Universal Robots PolyScope program: Main3.urp

Program Main3 (installation=main2 directory=/programs createdIn=5.11.5.1010327 lastSavedIn=5.11.5.1010327 robotSerialNumber=20215500677)
Calibrated DH parameters: a=[0.000204, -0.239222, -0.391845, -0.000001, 0.000022, 0]; d=[0.162722, -355.808559, 353.37206, 2.570385, 0.099741, 0.099629]; alpha=[1.571124, 0.000988, 0.008295, 1.568963, -1.570303, 0]; deltaTheta=[0, -0.973091, 7.204745, 0.05153, 0, 0]
Robot Program (runOnlyOnce=true)
  MoveJ speed 60 deg/s, acceleration 80 deg/s^2 (useActiveTCP=true) feature=CubeFront
    Waypoint Clear: TCP in base x=-162.331 y=-451.249 z=327.15 mm, rx=0.0678 ry=2.1899 rz=-2.19 rad; joints [27.656, -90.853, 115.036, 43.322, 49.382, -232.337] deg; TCP offset x=-1.34 y=-107.472 z=94.069 mm, rx=0.7854 ry=0 rz=0 rad; feature pose in base x=2.048 y=-607.004 z=173.227 mm, rx=-0.0204 ry=-2.2235 rz=-2.2094 rad
    Waypoint CubeOrigin: TCP in base x=2.125 y=-596.994 z=173.157 mm, rx=0.0109 ry=-2.2052 rz=2.2192 rad; joints [70.088, -70.787, 112.558, 4.336, 76.614, -194.298] deg
    Waypoint Clear: TCP in base x=-162.331 y=-451.249 z=327.15 mm, rx=0.0678 ry=2.1899 rz=-2.19 rad; joints [27.656, -90.853, 115.036, 43.322, 49.382, -232.337] deg
  MoveJ speed 60 deg/s, acceleration 80 deg/s^2 (useActiveTCP=false) tcp=pointer; feature=SandBack
    Waypoint Clear: TCP in base x=-162.331 y=-451.249 z=327.15 mm, rx=0.0678 ry=2.1899 rz=-2.19 rad; joints [27.656, -90.853, 115.036, 43.322, 49.382, -232.337] deg
    Waypoint CubeOrigin: TCP in base x=2.125 y=-596.994 z=173.157 mm, rx=0.0109 ry=-2.2052 rz=2.2192 rad; joints [70.088, -70.787, 112.558, 4.336, 76.614, -194.298] deg
    Waypoint Clear: TCP in base x=-162.331 y=-451.249 z=327.15 mm, rx=0.0678 ry=2.1899 rz=-2.19 rad; joints [27.656, -90.853, 115.036, 43.322, 49.382, -232.337] deg
